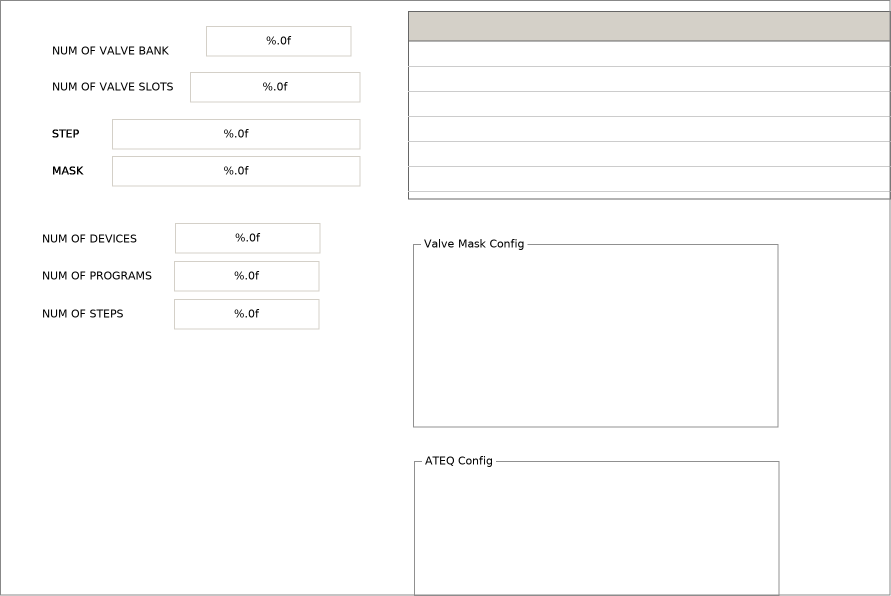
VISUALIZATION visMain  // 891x596
    Table (408,11 483x188), data array: GVL_VisVariable.anValveMask
        p3854506369: GVL_VisVariable.anValveMask[INDEX]
        p2232123230: GVL_visVariableMap.anValveMask[INDEX]
    Group (49,119 311x30)
        Textfield (63,0 248x30), "%.0f", text variable: GVL_VisVariable.visValveMaskIdx
            OnMouseClick: write GVL_VisVariable.visValveMaskIdx via VisuDialogs.Numpad
        Label (0,0 60x30), "STEP"
    Textfield (112,119 248x30), "%.0f", text variable: GVL_VisVariable.visValveMaskIdx
        OnMouseClick: write GVL_VisVariable.visValveMaskIdx via VisuDialogs.Numpad
    Label (49,119 60x30), "STEP"
    Textfield (112,119 248x30), "%.0f", text variable: GVL_VisVariable.visValveMaskIdx
        OnMouseClick: write GVL_VisVariable.visValveMaskIdx via VisuDialogs.Numpad
    Label (49,119 60x30), "STEP"
    Textfield (112,119 248x30), "%.0f", text variable: GVL_VisVariable.visValveMaskIdx
        OnMouseClick: write GVL_VisVariable.visValveMaskIdx via VisuDialogs.Numpad
    Label (49,119 60x30), "STEP"
    Group (49,156 311x30)
        Textfield (63,0 248x30), "%.0f", text variable: GVL_VisVariable.nValveMask
            OnMouseClick: write GVL_VisVariable.nValveMask via VisuDialogs.Numpad
        Label (0,0 60x30), "MASK"
    Textfield (112,156 248x30), "%.0f", text variable: GVL_VisVariable.nValveMask
        OnMouseClick: write GVL_VisVariable.nValveMask via VisuDialogs.Numpad
    Label (49,156 60x30), "MASK"
    Textfield (112,156 248x30), "%.0f", text variable: GVL_VisVariable.nValveMask
        OnMouseClick: write GVL_VisVariable.nValveMask via VisuDialogs.Numpad
    Label (49,156 60x30), "MASK"
    Textfield (112,156 248x30), "%.0f", text variable: GVL_VisVariable.nValveMask
        OnMouseClick: write GVL_VisVariable.nValveMask via VisuDialogs.Numpad
    Label (49,156 60x30), "MASK"
    GroupBox (413,236 365x191), "Valve Mask Config"
    Label (39,224 140x30), "NUM OF DEVICES"
    Textfield (174,261 145x30), "%.0f", text variable: nMaxProgramsToRun
        OnMouseClick: write nMaxProgramsToRun via Default, format %.0f
    Label (39,261 124x30), "NUM OF PROGRAMS"
    Textfield (174,299 145x30), "%.0f", text variable: nMaxTestSteps
        OnMouseClick: write nMaxTestSteps via Default, format %.0f
    Label (39,299 124x30), "NUM OF STEPS"
    GroupBox (414,453 365x143), "ATEQ Config"
    Label (49,36 141x30), "NUM OF VALVE BANK"
    Textfield (190,72 170x30), "%.0f", text variable: nMaxNumOfValveSlots
        OnMouseClick: write nMaxNumOfValveSlots via VisuDialogs.Numpad
    Label (49,72 141x30), "NUM OF VALVE SLOTS"
    Textfield (175,223 145x30), "%.0f", text variable: GVL_AteqConfig.nMaxDeviceCount
        OnMouseClick: write GVL_AteqConfig.nMaxDeviceCount via Default, format %.0f
    Textfield (206,26 145x30), "%.0f", text variable: GVL_ValveBankConfig.nMaxDeviceCount
        OnMouseClick: write GVL_ValveBankConfig.nMaxDeviceCount via Default, format %.0f
END_VISUALIZATION

(* stored: Version 1.1.0.1
   Visu visMain: Id {d1886aa2-3151-044a-2d27-02e663df3a34} *)
